// TIA Portal V17 export
// export: Created 2022-07-20T07:02:43.4977011Z, ExportSetting WithDefaults, DisplayName Totally Integrated Automation Portal, DisplayVersion V17, DisplayName TIA Portal Openness, DisplayVersion V17, DisplayName TIA Portal Version Control Interface, DisplayVersion V17, DisplayName SINAMICS Startdrive Advanced, DisplayVersion V17, DisplayName SINAMICS Startdrive G130, G150, S120, S150, SINAMICS MV, S210, DisplayVersion V17, DisplayName SINAMICS Startdrive G110M, G120, G120C, G120D, G120P, G115D, DisplayVersion V17, DisplayName STEP 7 Professional, DisplayVersion V17, DisplayName STEP 7 Safety, DisplayVersion V17, DisplayName WinCC Advanced, DisplayVersion V17
VAR_GLOBAL   // PLC tag table "Default tag table"
   clockInput AT %I0.0 : Bool;   // Clock generator input
   Tag_1 AT %ID1000 : DWord;
   Axe_1_Signal_A AT %Q0.2 : Bool;
   Axe_1_Signal_B AT %Q0.3 : Bool;
END_VAR
